# EPICS autosave request: galilDmc30017App/Db/galil_dmc30017_positions.req
# Save motor position
$(P)$(M).DVAL
